TYPE
    EtcSlaveBase_82538BE2 :
    STRUCT
    END_STRUCT
END_TYPE

(* stored: Version 1.1.0.1, ProductVersion 3.1.4024.12
   DUT EtcSlaveBase_82538BE2: Id {4b06efa6-f206-03bb-1d1b-80cdcbc0c201} *)
